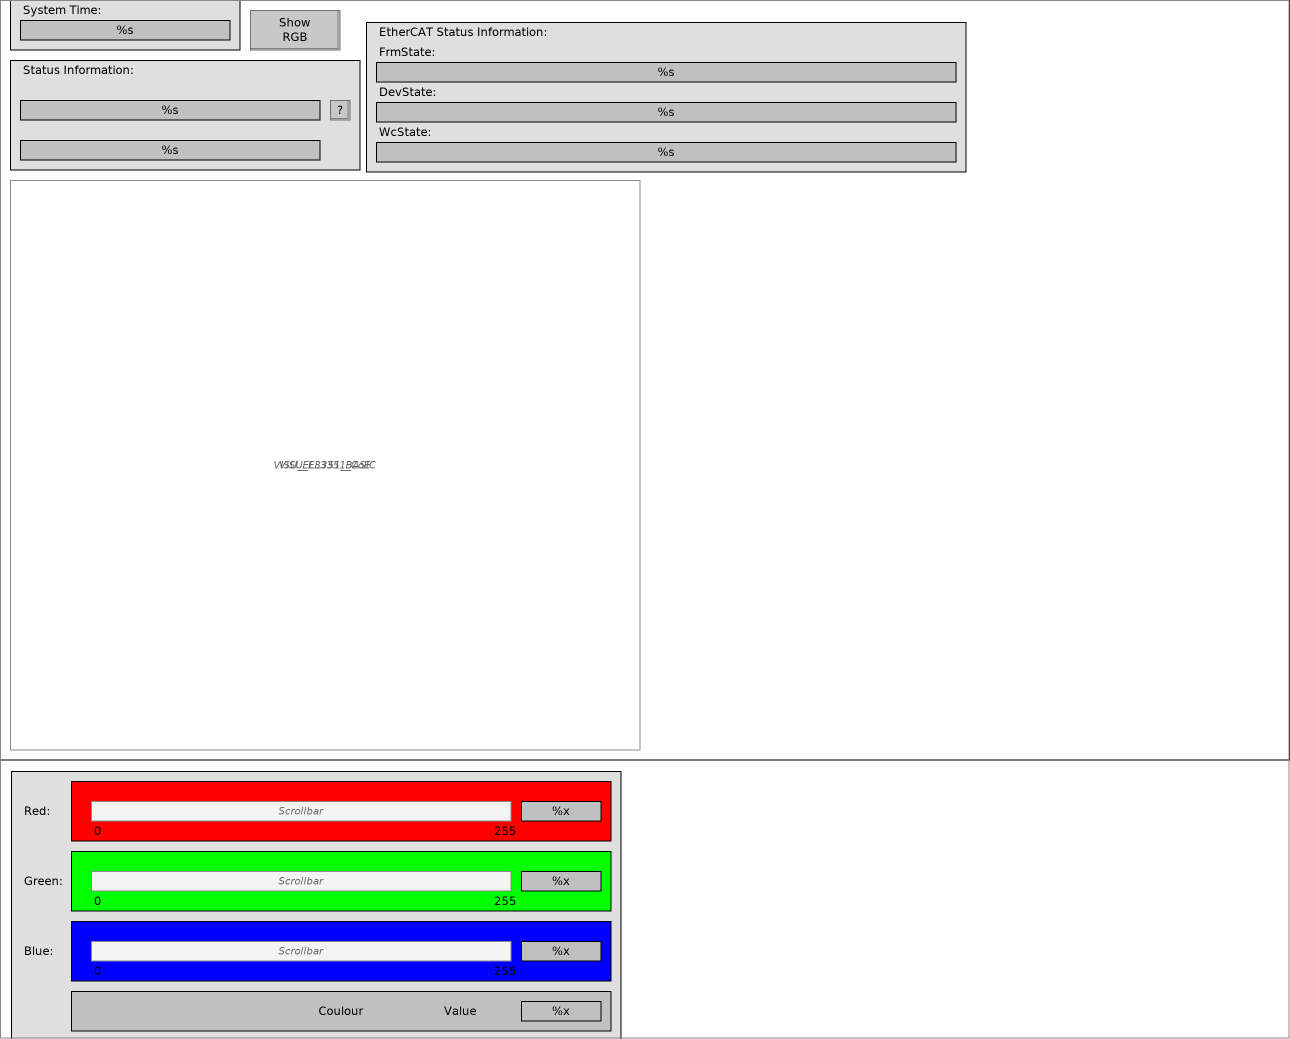
VISUALIZATION VSU_EL3351  // 1290x1039
    Rectangle (0,0 1290x760)
    Frame (10,180 630x570)
        shows VISU_EL3351_BASIC(m_Input_afbEL3351_Index_ := P_LoadCell.afbEL3351[1])
    Frame (10,180 630x570), invisible if: NOT P_LoadCell.afbEL3351[1].bVisuZoom
        shows VISU_EL3351_CoE(m_Input_afbEL3351_Index_ := P_LoadCell.afbEL3351[1])
    Rectangle (10,0 230x50)
    RoundedRectangle (20,20 210x20), "%s", text variable: P_LoadCell.fbGetTime.sDateAndTime
    Rectangle (20,0 100x20), "System Time:"
    Button (250,10 90x40), "Show RGB", pressed state: P_LoadCell.bShowRGB
        p3450524324: MAIN.dwButtonColour
        toggle P_LoadCell.bShowRGB
    Rectangle (370,41 460x130), "Placeholders are used to be able to have one visualization for each EL3351 that is connected. For every EL3351, a new visualization can be added and all placeholders for linked variables can be replaced by the new Instance. To do so, double klick on the visu, select "Placeholder" and choose a replacement for the placeholder afbEL3351[index]. To activate each visualization, click on "Enable". If just one EL3351 is connected, the 2nd visualization can stay disabled."
    Rectangle (10,60 350x110)
    Rectangle (20,60 150x20), "Status Information:"
    Rectangle (20,140 300x20), "%s", text variable: P_LoadCell.sAllTerminalsStatus, colour variable: P_LoadCell.dwAllTerminalsStatus
    Rectangle (20,100 300x20), "%s", text variable: P_LoadCell.sFieldBusStatus, colour variable: P_LoadCell.fbEtherCATDiagnosis.dwFieldbusStatus
    Group (366,22 598x148), invisible if: NOT P_LoadCell.bQuestionMarkFieldbusError
        Rectangle (0,0 600x150)
        Rectangle (10,0 210x20), "EtherCAT Status Information:"
        Rectangle (10,120 580x20), "%s", text variable: P_LoadCell.fbEtherCATDiagnosis.fbFrmWcStateDiagnosis.sFrmWcStateStatus, colour variable: P_LoadCell.fbEtherCATDiagnosis.fbFrmWcStateDiagnosis.dwFrmWcStateStatusColour
        Rectangle (10,40 580x20), "%s", text variable: P_LoadCell.fbEtherCATDiagnosis.fbFrmStateDiagnosis.sFrmStateStatus, colour variable: P_LoadCell.fbEtherCATDiagnosis.fbFrmStateDiagnosis.dwFrmStateStatusColour
        Rectangle (10,80 580x20), "%s", text variable: P_LoadCell.fbEtherCATDiagnosis.fbDevStateDiagnosis.sDevStateStatus, colour variable: P_LoadCell.fbEtherCATDiagnosis.fbDevStateDiagnosis.dwDevStateStatusColour
        Rectangle (10,20 160x20), "FrmState:"
        Rectangle (10,100 190x20), "WcState:"
        Rectangle (10,60 170x20), "DevState:"
    Group (11,771 608x268), invisible if: NOT P_LoadCell.bShowRGB
        Rectangle (0,0 610x270), invisible if: NOT P_LoadCell.bShowRGB
        Rectangle (60,10 540x60), invisible if: NOT P_LoadCell.bShowRGB
        Scrollbar (80,30 420x20), invisible if: NOT P_LoadCell.bShowRGB
            p1057716461: P_LoadCell.fbColours.byRed
        Rectangle (510,30 80x20), "%x", text variable: P_LoadCell.fbColours.byRed, invisible if: NOT P_LoadCell.bShowRGB
        Rectangle (10,30 70x20), "Red:", invisible if: NOT P_LoadCell.bShowRGB
        Rectangle (10,100 70x20), "Green:", invisible if: NOT P_LoadCell.bShowRGB
        Rectangle (60,80 540x60), invisible if: NOT P_LoadCell.bShowRGB
        Scrollbar (80,100 420x20), invisible if: NOT P_LoadCell.bShowRGB
            p1057716461: P_LoadCell.fbColours.byGreen
        Rectangle (510,100 80x20), "%x", text variable: P_LoadCell.fbColours.byGreen, invisible if: NOT P_LoadCell.bShowRGB
        Rectangle (10,170 70x20), "Blue:", invisible if: NOT P_LoadCell.bShowRGB
        Rectangle (60,150 540x60), invisible if: NOT P_LoadCell.bShowRGB
        Scrollbar (80,170 420x20), invisible if: NOT P_LoadCell.bShowRGB
            p1057716461: P_LoadCell.fbColours.byBlue
        Rectangle (510,170 80x20), "%x", text variable: P_LoadCell.fbColours.byBlue, invisible if: NOT P_LoadCell.bShowRGB
        RoundedRectangle (60,220 540x40), "Coulour", invisible if: NOT P_LoadCell.bShowRGB, colour variable: P_LoadCell.fbColours.dwColour
        Rectangle (80,50 30x20), "0", invisible if: NOT P_LoadCell.bShowRGB
        Rectangle (480,50 40x20), "255", invisible if: NOT P_LoadCell.bShowRGB
        Rectangle (80,190 30x20), "0", invisible if: NOT P_LoadCell.bShowRGB
        Rectangle (80,120 30x20), "0", invisible if: NOT P_LoadCell.bShowRGB
        Rectangle (480,190 40x20), "255", invisible if: NOT P_LoadCell.bShowRGB
        Rectangle (480,120 40x20), "255", invisible if: NOT P_LoadCell.bShowRGB
        Rectangle (510,230 80x20), "%x", text variable: P_LoadCell.fbColours.dwColour, invisible if: NOT P_LoadCell.bShowRGB
        Rectangle (430,230 70x20), "Value", invisible if: NOT P_LoadCell.bShowRGB
    Button (330,100 20x20), "?", pressed state: P_LoadCell.bQuestionMarkFieldbusError
        p3450524324: MAIN.dwButtonColour
        toggle P_LoadCell.bQuestionMarkFieldbusError
END_VISUALIZATION

(* stored: Version 1.1.0.1, ProductVersion 3.1.4024.12
   Visu VSU_EL3351: Id {0f4e4054-8c0d-43d4-b8b9-7fc9642185cd} *)
